PROGRAM MAIN
VAR

END_VAR

Axes();
Kinematics();
Home();
Singularity();

END_PROGRAM

(* stored: Version 1.1.0.1, ProductVersion 3.1.4018.9
   POU MAIN: Id {e9a9a825-28a7-4b93-8dd6-e16879b7ba33}, SpecialFunc None *)
